//-------------------------------------------------------------------------------------------//
//-------------------------------Desactivacion de los contactores----------------------------//
//-------------------------------------------------------------------------------------------//
gSalidasPLC.Contactor := FALSE;
gSalidasPLC.Contactor2 := FALSE;

//-------------------------------------------------------------------------------------------//
//-----------Desactivacion del eletrofreno y de los canales del relé de seguridad------------//
//-------------------------------------------------------------------------------------------//
gSalidasPLC.Eletrofreno := FALSE;
gSalidasPLC.Ch1_ReleSeguridad := FALSE;
gSalidasPLC.Ch2_ReleSeguridad := FALSE;

//-------------------------------------------------------------------------------------------//
//-------------------Desactivacion del contactopr que habilita el variador-------------------//
//-------------------------------------------------------------------------------------------//
gSalidasPLC.ContactorHabVariador := FALSE;

END_PROGRAM

// StandardPLC/Application/CÓDIGO/Sub Dispositivos/DISP02_Indicadores
PROGRAM DISP02_Indicadores
VAR_INPUT
	I_SeleccionModo 		:BYTE;
END_VAR
VAR_OUTPUT
	O_IndicadorRojo			:BOOL;
	O_IndicadoAmarillo		:BOOL;
	O_IndicadoVerde			:BOOL;
	O_IndicadoAcustico		:BOOL;
END_VAR
VAR
	TON_Tren1sA				:BOOL;
	TON_Tren1s				:TON;
	TOF_Tren1s				:TON;
	
	TON_Automatico			:TON;
	TOF_Automatico			:TON;

	SecuenciaEncendido 		:BYTE;
END_VAR

(*//////////////////////////////////////////////////////////////////////////////////////////////////////////////////////////////////////////////////////////////////////////////////////////////////////////////////////////////////////////////////
DISP02_Indicadores (PRG)                     

Description:	Bloque control señales lumínicas y acústicas
				 
///////////////////////////////////////////////////////////////////////////////////////////////////////////////////////////////////////////////////////////////////////////////////////////////////////////////////////////////////////////////////// *)

TON_Tren1s( IN:=TOF_Tren1s.Q, PT:=T#500ms);
TOF_Tren1s( IN:=( NOT TON_Tren1s.Q ), PT:=T#500MS);

TON_Automatico( IN:=TOF_Automatico.Q, PT:=T#1S);
TOF_Automatico( IN:=( NOT TON_Automatico.Q ), PT:=T#1S);

CASE I_SeleccionModo OF
	0: (*Secuencia encendido*)
		CASE SecuenciaEncendido OF
			0:
				IF TON_Tren1s.Q<>TON_Tren1sA THEN SecuenciaEncendido := 1; END_IF;
				O_IndicadorRojo := 1;		O_IndicadoAcustico := 1;
				O_IndicadoAmarillo := 0;	O_IndicadoVerde := 0;
			1:
				IF TON_Tren1s.Q<>TON_Tren1sA THEN SecuenciaEncendido := 2; END_IF;
				O_IndicadorRojo := 0;		O_IndicadoAcustico := 0;
				O_IndicadoAmarillo := 1;	O_IndicadoVerde := 0;
			2:
				IF TON_Tren1s.Q<>TON_Tren1sA THEN SecuenciaEncendido := 0; END_IF;
				O_IndicadorRojo := 0;		O_IndicadoAcustico := 0;
				O_IndicadoAmarillo := 0;	O_IndicadoVerde := 1;
		END_CASE;
		TON_Tren1sA  := TON_Tren1s.Q;

	1:	O_IndicadoVerde := TOF_Tren1s.Q;   //----- Estado espera inicio	-----//	
		O_IndicadoAmarillo := 0;						
		O_IndicadorRojo := 0;						
		O_IndicadoAcustico := 0;		
		
	2:	O_IndicadoVerde := 1;		       //----- Estado reposo -----//			
		O_IndicadoAmarillo := 0;						
		O_IndicadorRojo := 0;						
		O_IndicadoAcustico := 0;		

	3:	O_IndicadoVerde := 0;			  //----- Ejecutando acción automático -----//		
		O_IndicadoAmarillo := TOF_Automatico.Q;						
		O_IndicadorRojo := 0;						
		O_IndicadoAcustico := TOF_Automatico.Q;		

	4:	O_IndicadoVerde := 0;			  //----- Ejecutando acción - pausa -----//	
		O_IndicadoAmarillo := TOF_Tren1s.Q;		
		O_IndicadorRojo := 0;						
		O_IndicadoAcustico := 0;		
 
	5:	O_IndicadoVerde := 0;	         //----- Manual/Degradado -----//					
		O_IndicadoAmarillo := TOF_Tren1s.Q;		
		O_IndicadorRojo := TOF_Tren1s.Q;		
		O_IndicadoAcustico := 0;		

	6:	O_IndicadoVerde := 0;		     //----- Anomalia ADVERTENCIA autorearmable -----//				
		O_IndicadoAmarillo := 0;						
		O_IndicadorRojo := 1;						
		O_IndicadoAcustico := TOF_Tren1s.Q;	

	7:	O_IndicadoVerde := 0;			 //----- Anomalia ADVERTENCIA rearmable	-----//		
		O_IndicadoAmarillo := 0;						
		O_IndicadorRojo := TOF_Tren1s.Q;		
		O_IndicadoAcustico := TOF_Tren1s.Q;

	8:	O_IndicadoVerde := 0;		     //----- Anomalia CRÍTCA/FATAL activa -----//				
		O_IndicadoAmarillo := 0;						
		O_IndicadorRojo := TOF_Tren1s.Q;		
		O_IndicadoAcustico := 1;		

	9:	O_IndicadoVerde := 0;		     //----- Anomalia FATAL pausa -----//				
		O_IndicadoAmarillo := 0;						
		O_IndicadorRojo := 1;						
		O_IndicadoAcustico := 0;		

	10:	O_IndicadoVerde := 0;			//----- Anomalia SEVERA activa - requiere posicion segura -----//	
		O_IndicadoAmarillo := TOF_Tren1s.Q;		
		O_IndicadorRojo := 1;						
		O_IndicadoAcustico := TOF_Tren1s.Q;

	11:	O_IndicadoVerde := 0;		    //----- Anomalia SEVERA pausa - requiere posicion segura -----//		
		O_IndicadoAmarillo := TOF_Tren1s.Q;		
		O_IndicadorRojo := 1;						
		O_IndicadoAcustico := 0;
		
	12: O_IndicadoVerde := 0;			//----- Anomalia SEVERA activa - requiere posicion segura -----//	
		O_IndicadoAmarillo := 0;		
		O_IndicadorRojo := TOF_Tren1s.Q;						
		O_IndicadoAcustico := TOF_Tren1s.Q;
		
	13: O_IndicadoVerde := 0;			//----- Parpadeo de cuando se pulsa Seta -----//	
		O_IndicadoAmarillo := 0;		
		O_IndicadorRojo := 1;						
		O_IndicadoAcustico := 1;
		
	14: O_IndicadoVerde := 0;			//----- Parpadeo de cuando desenclavamos seta -----//	
		O_IndicadoAmarillo := TOF_Tren1s.Q;		
		O_IndicadorRojo := TOF_Tren1s.Q;						
		O_IndicadoAcustico := 0;
		
	15: O_IndicadoVerde := 1;			//----- Parpadeo de cuando desenclavamos seta -----//	
		O_IndicadoAmarillo := 0;		
		O_IndicadorRojo := 0;						
		O_IndicadoAcustico := 1;
END_CASE;

END_PROGRAM

// StandardPLC/Application/CÓDIGO/Sub Temporizacion/TEMP00_TiempoInicio
PROGRAM TEMP00_TiempoInicio
VAR_INPUT
	I_TiempoEncendido		:INT;
END_VAR
VAR_OUTPUT
	O_FinTiempo				:BOOL;
END_VAR
VAR
	Primera					:BOOL := TRUE;
	SegundosEncendido		:INT;
	Tren500msA				:BOOL;
	TON_Tren500ms 			:TON;
	TOF_Tren500ms			:TOF;
END_VAR

(*/////////////////////////////////////////////////////////////////////////////////////////////////////////////////////////////////////////////////////////////////////////////////////////////////////////////////////////////////////////////////
TEMP00_TiempoInicio (PRG)                     

Description:  Módulo encargado de realizar la cuenta atrás de inicio.
			  I_TiempoEncendido: cantidad entera de segundos que deseamos como inicio.
			  O_FinTiempo: TRUE si cuenta a llegado a su fin. FALSE en otro caso.				
				 
///////////////////////////////////////////////////////////////////////////////////////////////////////////////////////////////////////////////////////////////////////////////////////////////////////////////////////////////////////////////////// *)

TON_Tren500ms( IN:=TOF_Tren500ms.Q, PT:=T#500ms);
TOF_Tren500ms( IN:=( NOT TON_Tren500ms.Q ), PT:=T#500ms);

IF Primera THEN
	SegundosEncendido := I_TiempoEncendido;
	Primera := FALSE;
ELSE
	IF ( (SegundosEncendido>0) AND TON_Tren500ms.Q AND (NOT Tren500msA) ) THEN
		SegundosEncendido := SegundosEncendido -1;
	END_IF;
END_IF;

Tren500msA := TON_Tren500ms.Q;
O_FinTiempo := (SegundosEncendido=0);

END_PROGRAM

// Project Information/GetNumberProperty
// This function has been automatically generated from the project information.
{attribute 'signature_flag' := '1073741824'}
{attribute 'register_in_runtime'}
FUNCTION GetNumberProperty : DINT
VAR_INPUT
	stKey: WSTRING;
END_VAR

GetNumberProperty := 0;

END_FUNCTION

// Project Information/GetVersionProperty
// This function has been automatically generated from the project information.
{attribute 'signature_flag' := '1073741824'}
{attribute 'register_in_runtime'}
FUNCTION GetVersionProperty : VERSION
VAR_INPUT
	stKey: WSTRING;
END_VAR

IF stKey = "Version" THEN
	GetVersionProperty.uiMajor := 2;
	GetVersionProperty.uiMinor := 4;
	GetVersionProperty.uiServicePack := 13;
	GetVersionProperty.uiPatch := 0;
ELSE
	GetVersionProperty.uiMajor := 0;
	GetVersionProperty.uiMinor := 0;
	GetVersionProperty.uiServicePack := 0;
	GetVersionProperty.uiPatch := 0;
END_IF

END_FUNCTION

// Project Information/GetBooleanProperty
// This function has been automatically generated from the project information.
{attribute 'signature_flag' := '1073741824'}
{attribute 'register_in_runtime'}
FUNCTION GetBooleanProperty : BOOL
VAR_INPUT
	stKey: WSTRING;
END_VAR

IF stKey = "Released" THEN
	GetBooleanProperty := FALSE;
ELSE
	GetBooleanProperty := FALSE;
END_IF

END_FUNCTION

// Project Information/GetTextProperty
// This function has been automatically generated from the project information.
{attribute 'signature_flag' := '1073741824'}
{attribute 'register_in_runtime'}
FUNCTION GetTextProperty : WSTRING
VAR_INPUT
	stKey: WSTRING;
END_VAR

IF stKey = "Company" THEN
	GetTextProperty := "ifm electronic";
ELSIF stKey = "Description" THEN
	GetTextProperty := "Project template with CR711S configured 2.25MByte Standard 2.25MByte Safety";
ELSIF stKey = "Project" THEN
	GetTextProperty := "SUZUKI";
ELSIF stKey = "Title" THEN
	GetTextProperty := "ifmCR711S_TemplateProject";
ELSE
	GetTextProperty := "";
END_IF

END_FUNCTION

// Project Information/GetTextProperty2
// This function has been automatically generated from the project information.
{attribute 'signature_flag' := '1073741824'}
{attribute 'register_in_runtime'}
FUNCTION GetTextProperty2 : POINTER TO WSTRING
VAR_INPUT
	stKey: WSTRING;
END_VAR

IF stKey = "Company" THEN
	GetTextProperty2 := ADR("ifm electronic");
ELSIF stKey = "Description" THEN
	GetTextProperty2 := ADR("Project template with CR711S configured 2.25MByte Standard 2.25MByte Safety");
ELSIF stKey = "Project" THEN
	GetTextProperty2 := ADR("SUZUKI");
ELSIF stKey = "Title" THEN
	GetTextProperty2 := ADR("ifmCR711S_TemplateProject");
ELSE
	GetTextProperty2 := ADR("");
END_IF

END_FUNCTION

// Project Information/GetTitle
// This function has been automatically generated from the project information.
{attribute 'signature_flag' := '1073741824'}
{attribute 'register_in_runtime'}
FUNCTION GetTitle : WSTRING
VAR_INPUT
	
END_VAR

GetTitle := "ifmCR711S_TemplateProject";

END_FUNCTION

// Project Information/GetCompany
// This function has been automatically generated from the project information.
{attribute 'signature_flag' := '1073741824'}
{attribute 'register_in_runtime'}
FUNCTION GetCompany : WSTRING
VAR_INPUT
	
END_VAR

GetCompany := "ifm electronic";

END_FUNCTION

// Project Information/GetVersion
// This function has been automatically generated from the project information.
{attribute 'signature_flag' := '1073741824'}
{attribute 'register_in_runtime'}
FUNCTION GetVersion : VERSION
VAR_INPUT
	
END_VAR

GetVersion.uiMajor := 2;
GetVersion.uiMinor := 4;
GetVersion.uiServicePack := 13;
GetVersion.uiPatch := 0;

END_FUNCTION

// StandardPLC/Application/CÓDIGO/AUX_IFM/fb_OutputAnaAddConf_sp_ST_V02
FUNCTION_BLOCK fb_OutputAnaAddConf_sp_ST_V02
VAR_INPUT
	IN_ResetError:BOOL;	
	IN_uiChannel:UINT;
	IN_eModeChannel:ifmIOcommon.MODE_OUTPUT;	
	IN_eDestination:ifmIOconfigDiagProt.DEST;
	IN_eDiagMode:ifmIOconfigDiagProt.eDIAG_PROT_MODE;
	IN_DetectionTime:UINT;
	IN_DiagLimMin:UINT;
	IN_DiagLimMax:UINT;

	IN_uiValue:UINT;
	
		
END_VAR
	
VAR_OUTPUT
	OUT_Done:BOOL;
	OUT_Error:BOOL;
	OUT_DiagInfo:ifmTypes.DIAG_INFO;	
	OUT_DiagInfoProt: ifmTypes.DIAG_INFO;
	OUT_DiagInfoLevel: ifmTypes.DIAG_INFO;	
END_VAR
VAR
	
	l_xExecute:BOOL;
	ConfigDiagLevel: ifmIOconfigDiagProt.ConfigDiagLevel;
	ConfigDiagProt: ifmIOconfigDiagProt.ConfigDiagProt;

	l_xExecute_DiagLevel:BOOL;
	l_xExecuted_DiagLevel:BOOL;	
	l_xExecute_DiagProt:BOOL;
	l_xExecuted_DiagProt:BOOL;
	R_TRIG_Execute: R_TRIG;
	Output:ifmIOcommon.Output;
	R_TRIG_Done: R_TRIG;
END_VAR
VAR // added by the converter: edge detectors and wires of the graphical bodies
    _w1 : BOOL;
END_VAR

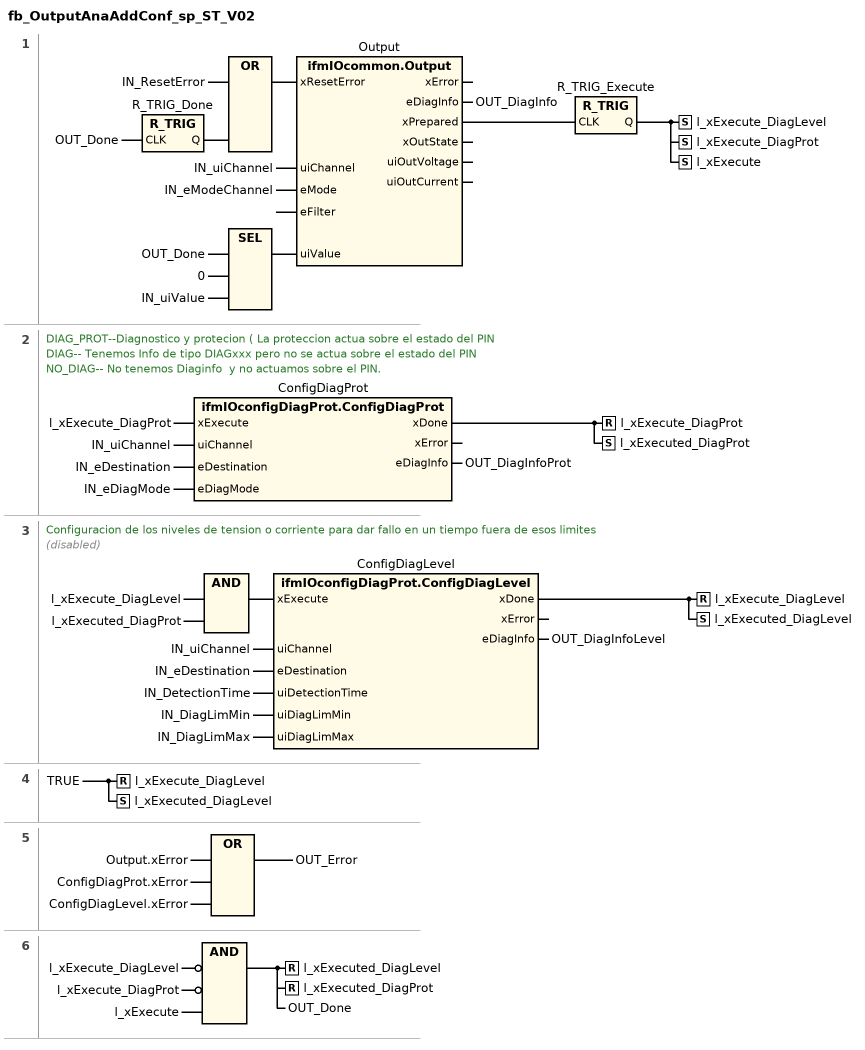
// NETWORK 1
R_TRIG_Done(CLK := OUT_Done); // R_TRIG
Output(
    xResetError := IN_ResetError OR R_TRIG_Done.Q,
    uiChannel := IN_uiChannel,
    eMode := IN_eModeChannel,
    uiValue := SEL(OUT_Done, 0, IN_uiValue),
    eDiagInfo => OUT_DiagInfo); // ifmIOcommon.Output
R_TRIG_Execute(CLK := Output.xPrepared); // R_TRIG
l_xExecute_DiagLevel S= R_TRIG_Execute.Q;
l_xExecute_DiagProt S= R_TRIG_Execute.Q;
l_xExecute S= R_TRIG_Execute.Q;

// NETWORK 2
// DIAG_PROT--Diagnostico y protecion ( La proteccion actua sobre el estado del PIN
// DIAG-- Tenemos Info de tipo DIAGxxx pero no se actua sobre el estado del PIN
// NO_DIAG-- No tenemos Diaginfo  y no actuamos sobre el PIN.
ConfigDiagProt(
    xExecute := l_xExecute_DiagProt,
    uiChannel := IN_uiChannel,
    eDestination := IN_eDestination,
    eDiagMode := IN_eDiagMode,
    eDiagInfo => OUT_DiagInfoProt); // ifmIOconfigDiagProt.ConfigDiagProt
l_xExecute_DiagProt R= ConfigDiagProt.xDone;
l_xExecuted_DiagProt S= ConfigDiagProt.xDone;

// NETWORK 3 (disabled)
// Configuracion de los niveles de tension o corriente para dar fallo en un tiempo fuera de esos limites
// ConfigDiagLevel(
//     xExecute := l_xExecute_DiagLevel AND l_xExecuted_DiagProt,
//     uiChannel := IN_uiChannel,
//     eDestination := IN_eDestination,
//     uiDetectionTime := IN_DetectionTime,
//     uiDiagLimMin := IN_DiagLimMin,
//     uiDiagLimMax := IN_DiagLimMax,
//     eDiagInfo => OUT_DiagInfoLevel); // ifmIOconfigDiagProt.ConfigDiagLevel
// l_xExecute_DiagLevel R= ConfigDiagLevel.xDone;
// l_xExecuted_DiagLevel S= ConfigDiagLevel.xDone;

// NETWORK 4
l_xExecute_DiagLevel R= TRUE;
l_xExecuted_DiagLevel S= TRUE;

// NETWORK 5
OUT_Error := Output.xError OR ConfigDiagProt.xError OR ConfigDiagLevel.xError;

// NETWORK 6
_w1 := NOT l_xExecute_DiagLevel AND NOT l_xExecute_DiagProt AND l_xExecute;
l_xExecuted_DiagLevel R= _w1;
l_xExecuted_DiagProt R= _w1;
OUT_Done := _w1;

END_FUNCTION_BLOCK
